FUNCTION_BLOCK FB_Valve_2_10V IMPLEMENTS I_Valve
VAR_INPUT
END_VAR
VAR_OUTPUT
END_VAR
VAR
	fValSet		:	REAL;
	nValSetRaw	AT %Q*	:	INT;
	fValAct		:	REAL;
	nValActRaw	AT %I*	:	INT;
	
	nIntMin		:	INT	:=	6553;
	nIntMax		:	INT	:=	32767;
	
	//Error detection
	bErr	:	BOOL;
	MaxTime	:	TIME	:=	T#1M;	//Maximum time to allow for movement
	MaxDiff	:	REAL	:=	5;		//Maximum percentage difference
	TimED	:	TON;
END_VAR

PROPERTY Error : BOOL
GET
Error := bErr;
END_GET
SET
bErr := Error;
END_SET
END_PROPERTY

PROPERTY OpenPercAct : REAL
GET
OpenPercAct	:=	fValAct;
END_GET
SET
fValAct	:=	OpenPercAct;
END_SET
END_PROPERTY

PROPERTY OpenPercSet : REAL
GET
OpenPercSet := fValSet;
END_GET
SET
fValSet := OpenPercSet;
END_SET
END_PROPERTY

METHOD Run : BOOL
IF fValSet < 0 THEN
	nValSetRaw	:=	0;
ELSE
	nValSetRaw := REAL_TO_INT(nIntMin + (fValSet/100)*(nIntMax-nIntMin));
END_IF

IF nValActRaw < 100 THEN
	fValAct := 0;
ELSE
	fValAct := 100*INT_TO_REAL(nValActRaw-nIntMin)/(nIntMax-nIntMin); //0-100% between Min and Max
END_IF

//Error detection
IF ABS(fValSet - fValAct) > MaxDiff THEN
	TimED(IN:=TRUE,PT:=MaxTime);
	IF TimED.Q THEN
		bErr	:=	TRUE;
	END_IF
ELSE
	TimED(In:=FALSE);
	bErr	:=	FALSE;
END_IF
END_METHOD

END_FUNCTION_BLOCK

(* stored: Version 1.1.0.1, ProductVersion 3.1.4022.10
   POU FB_Valve_2_10V: Id {3d6f0c4c-7091-433d-9206-ca167187df45}, SpecialFunc None
   Property Error: Id {c64f3baa-2842-4663-8dc7-d4d6876f1ac2}
   Get Get: Id {e3241b09-0eb7-44db-b486-2f179656e658}
   Set Set: Id {ff13ee99-0c04-42d3-b2a6-250c9c15b27e}
   Property OpenPercAct: Id {89e5fad3-85b4-4451-92dc-e91e994a45cf}
   Get Get: Id {333363fe-f4bc-4c70-8dbd-e3235597e1e9}
   Set Set: Id {f306478a-4dcb-43ca-9c9a-6c27bbaa3b05}
   Property OpenPercSet: Id {4d8785bc-ec30-433f-bf34-36204ffce037}
   Get Get: Id {c05774ab-866d-4582-a095-ec10c1450998}
   Set Set: Id {2df06ab4-5b5a-4e7a-a78d-a1438ccdef8e}
   Method Run: Id {383d8f0a-acf2-43b9-89c8-e35835787764} *)
